SUBAPPLICATION WaitForConnection (* Subapplication Type *)
  (* Standard: 61499-2; Description: Copyright (c) 2019 fortiss GmbH This program and the accompanying materials are made SPDX-License-Identifier: EPL-2.0 *)
  (* Version 1.0, 2020-04-15, Jose Cabral, fortiss GmbH *)
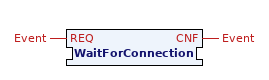
  EVENT_INPUT
    REQ;
  END_EVENT
  EVENT_OUTPUT
    CNF;
  END_EVENT
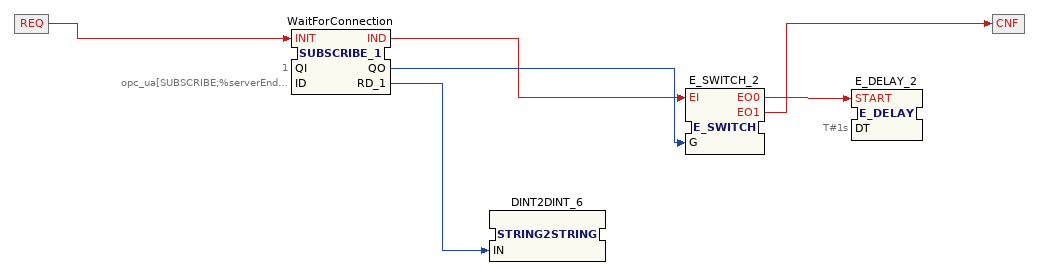
  FBS
    E_SWITCH_2 : E_SWITCH;
    DINT2DINT_6 : STRING2STRING;
    E_DELAY_2 : E_DELAY(DT := T#1s);
    WaitForConnection : SUBSCRIBE_1(QI := 1, ID := opc_ua[SUBSCRIBE;%serverEndpoint%; %connectionTesterNode%]);
  END_FBS
  EVENT_CONNECTIONS
    E_SWITCH_2.EO0 TO E_DELAY_2.START;
    E_SWITCH_2.EO1 TO CNF;
    REQ TO WaitForConnection.INIT;
    WaitForConnection.IND TO E_SWITCH_2.EI;
  END_CONNECTIONS
  DATA_CONNECTIONS
    WaitForConnection.QO TO E_SWITCH_2.G;
    WaitForConnection.RD_1 TO DINT2DINT_6.IN;
  END_CONNECTIONS
END_SUBAPPLICATION
